(* PLC project Unnamed, Unknown Unnamed 1 *)
(* stored: creationDateTime 2025-06-13T19:18:38, modificationDateTime 2025-06-13T21:31:00 *)

PROGRAM part4
  VAR
    main_sw_btn AT %IX0.0 : BOOL;
    car_sensor_1 AT %IX0.1 : BOOL;
    car_sensor_2 AT %IX0.2 : BOOL;
    green_entr_light AT %QX0.0 : BOOL;
    greep_pkg_light AT %QX0.1 : BOOL;
    red_entr_light AT %QX0.2 : BOOL;
    red_pkg_light AT %QX0.3 : BOOL;
    main_sw_indicator AT %QX0.4 : BOOL;
  END_VAR
  VAR
    state : UINT := 0;
    state_system_off : UINT := 0;
    state_no_cars : UINT := 1;
    state_car_entering : UINT := 2;
    state_car_exiting : UINT := 3;
    system_off : BOOL;
    no_cars : BOOL;
    car_entering : BOOL;
    car_exiting : BOOL;
    broken : BOOL;
    CTUD0 : CTUD;
    TP0 : TP;
  END_VAR
  VAR  (* added by the conversion: wires and edge detectors of the diagram *)
    F_TRIG1 : F_TRIG;
    F_TRIG2 : F_TRIG;
    R_TRIG3 : R_TRIG;
    R_TRIG4 : R_TRIG;
    R_TRIG5 : R_TRIG;
    R_TRIG6 : R_TRIG;
  END_VAR

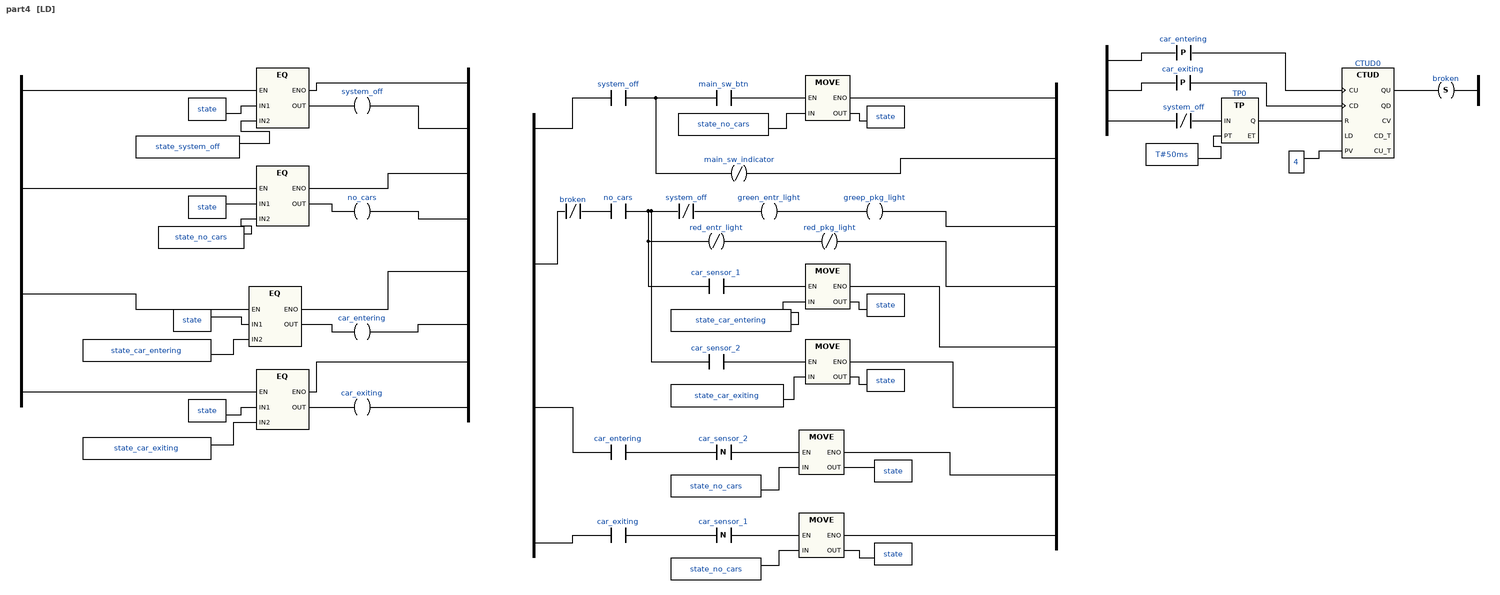
(* LD diagram, written out as Structured Text *)
no_cars := state = state_no_cars;
car_entering := state = state_car_entering;
system_off := state = state_system_off;
car_exiting := state = state_car_exiting;
IF system_off AND main_sw_btn THEN state := state_no_cars; END_IF;
main_sw_indicator := NOT system_off;
green_entr_light := NOT broken AND no_cars AND NOT system_off;
greep_pkg_light := NOT broken AND no_cars AND NOT system_off;
IF NOT broken AND no_cars AND car_sensor_1 THEN state := state_car_entering; END_IF;
IF NOT broken AND no_cars AND car_sensor_2 THEN state := state_car_exiting; END_IF;
F_TRIG1(CLK := car_sensor_2);
IF car_entering AND F_TRIG1.Q THEN state := state_no_cars; END_IF;
F_TRIG2(CLK := car_sensor_1);
IF car_exiting AND F_TRIG2.Q THEN state := state_no_cars; END_IF;
red_entr_light := NOT (NOT broken AND no_cars);
red_pkg_light := NOT (NOT broken AND no_cars);
R_TRIG3(CLK := car_entering);
R_TRIG4(CLK := R_TRIG3.Q);
R_TRIG5(CLK := car_exiting);
R_TRIG6(CLK := R_TRIG5.Q);
TP0(IN := NOT system_off, PT := T#50ms);
CTUD0(CU := R_TRIG4.Q, CD := R_TRIG6.Q, R := TP0.Q, PV := 4);
IF CTUD0.QU THEN broken := TRUE; END_IF;
END_PROGRAM

CONFIGURATION Config0
  RESOURCE Res0 ON PLC
    TASK task0(INTERVAL := T#20ms, PRIORITY := 0);
    PROGRAM instance0 WITH task0 : part4;
  END_RESOURCE
END_CONFIGURATION
